TYPE ExampleDomain_Hmi :
STRUCT
	sStatusText			: Str;
END_STRUCT
END_TYPE

(* stored: Version 1.1.0.1
   DUT ExampleDomain_Hmi: Id {6b406949-ad69-468f-91b7-41a3d28dbbaa} *)
